TYPE DoChannelTriState :
STRUCT
	{attribute addProperty Name "Output"}
	Output AT %Q* : BOOL;
	{attribute addProperty Name "TriState"}
	TriState AT %Q* : BOOL;
END_STRUCT
END_TYPE

(* stored: Version 1.1.0.1, ProductVersion 3.1.4024.9
   DUT DoChannelTriState: Id {f2df484e-c6bd-0755-129e-bbe56e8ea1a1} *)
